METHOD contains : BOOL //check contents, not pointer value
VAR_INPUT
	value : REFERENCE TO AdsMessage;
END_VAR
VAR_OUTPUT
	atIndex : INT;
END_VAR
VAR
	temp : REFERENCE TO AdsMessage;
	i : INT;
END_VAR
IF length = 0 THEN
	contains := FALSE;
	RETURN;
END_IF

FOR i:=0 TO length-1 BY 1 DO
	temp := get(index := i, getSize => );
	
	IF 
		SIZEOF(value) = entrySize AND //same size
		MEMCMP(ADR(temp), ADR(value), SIZEOF(entrySize)) = 0 //same data
	THEN
		contains := TRUE;
		atIndex := i;
		RETURN;
	END_IF
	
END_FOR
contains := FALSE;
END_METHOD

METHOD get : REFERENCE TO AdsMessage
VAR_INPUT
	index : INT;
END_VAR
VAR_OUTPUT
	getSize : UDINT;
	ok : BOOL;
END_VAR
VAR
	temp : POINTER TO AdsMessage;
END_VAR
IF
	length = 0 OR
	index < 0 OR
	index >= length
THEN
	RETURN;
END_IF

ok := elements.GetEntry(diIndex := index, pResultEntry := ADR(temp));
get REF= temp^;

getSize := SIZEOF(get);
END_METHOD

METHOD isEmpty : BOOL
VAR_INPUT
END_VAR
isEmpty := length = 0;
END_METHOD

METHOD poll : AdsMessage
VAR_OUTPUT
	getSize : ULINT;
END_VAR
VAR
	tempRef : REFERENCE TO AdsMessage;
	tempPtr : POINTER TO AdsMessage;
END_VAR
IF length > 0 THEN
	tempRef REF= get(index := 0, getSize => getSize);
	//poll := get(index := 0, getSize => getSize);
	poll := tempRef;
	
	tempPtr := ADR(tempRef);
	__DELETE(tempPtr);
	
	elements.RemoveEntry(diIndex := 0);
	
	length := length - 1;
END_IF
END_METHOD

METHOD push : BOOL
VAR_INPUT
	value : REFERENCE TO AdsMessage;
END_VAR
VAR
	temp : POINTER TO AdsMessage;
END_VAR
IF length < maxElements THEN
	temp := __NEW(AdsMessage);
	temp^ := value;
	
	push := elements.AddEntryPtr(pEntry := temp);
	
	length := length + 1;
END_IF
END_METHOD

METHOD set : BOOL
VAR_INPUT
	i : INT;
	value : REFERENCE TO AdsMessage;
END_VAR
VAR
	temp : REFERENCE TO AdsMessage;
END_VAR
IF length = 0 THEN
	RETURN;
END_IF

IF i >= 0 AND i < length THEN
	temp REF= get(i);
	temp := value;
	
	set := TRUE;
END_IF
END_METHOD

{attribute 'call_after_init'}
METHOD setup : BOOL
VAR_INPUT
END_VAR
entrySize := SIZEOF(AdsMessage);

clear();
END_METHOD

METHOD size : INT
size := length;
END_METHOD

END_FUNCTION_BLOCK

// ---- DUTs/Hardware/Conveyors/ConveyorSC_NC.TcPOU
FUNCTION_BLOCK ConveyorSC_NC
VAR_INPUT
	bEnable : BOOL;
END_VAR
VAR_OUTPUT
	sensorEntry AT %I* : BOOL := TRUE;
	sensorExit AT %I* : BOOL;
	
	trueMode : ConveyorMode;
	requestedMode : ConveyorMode;
	
	position : LREAL;
	velocity : LREAL;
	ready : BOOL;
	error : BOOL;
END_VAR
VAR
	axis : AXIS_REF;
	
	mcReadPosition : MC_ReadActualPosition; //continuous enable FBs
	mcReadVelocity : MC_ReadActualVelocity;
	mcReadError : MC_ReadAxisError;
	mcPower : MC_Power;
	
	mcReset : MC_Reset; //rising edge FBs
	mcMoveAbsolute : MC_MoveAbsolute;
	mcMoveRelative : MC_MoveRelative;
	mcMoveVelocity : MC_MoveVelocity;
	
	mcSetPosition : MC_SetPosition;
	mcStop : MC_Stop;
END_VAR
VAR_STAT CONSTANT
	targetingVelocity : INT := 500;
	continuousVelocity : INT := 100;
END_VAR
(*
standard slat conveyor - no lifter
compliant with PLCopen motion control
*)

blocks();

mcReset.Execute := FALSE;
mcMoveAbsolute.Execute := FALSE;
mcMoveRelative.Execute := FALSE;
mcMoveVelocity.Execute := FALSE;
mcSetPosition.Execute := FALSE;
mcStop.Execute := FALSE;

blocks();

PROPERTY Active : BOOL
GET
Active := 
	mcMoveAbsolute.Busy OR 
	mcMoveRelative.Busy OR 
	mcMoveVelocity.Busy OR 
	mcSetPosition.Busy OR 
	mcReset.Busy OR 
	mcStop.Busy;
END_GET
END_PROPERTY

METHOD PRIVATE blocks : BOOL
mcReadPosition(
	Axis:= axis, 
	Enable:= TRUE, 
	Valid=> , 
	Busy=> , 
	Error=> , 
	ErrorID=> , 
	Position=> position);
	
mcReadVelocity(
	Axis:= axis, 
	Enable:= TRUE, 
	Valid=> , 
	Busy=> , 
	Error=> , 
	ErrorID=> , 
	ActualVelocity=> velocity);
	
mcReadError(
	Axis:= axis, 
	Enable:= TRUE, 
	Valid=> , 
	Busy=> , 
	Error=> , 
	ErrorID=> , 
	AxisErrorID=> );

mcReset(
	Axis:= axis, 
	Execute:= , 
	Done=> , 
	Busy=> , 
	Error=> , 
	ErrorID=> );

mcPower(
	Axis:= axis, 
	Enable:= bEnable, 
	Enable_Positive:= TRUE, 
	Enable_Negative:= TRUE, 
	Override:= 100, 
	BufferMode:= , 
	Options:= , 
	Status=> , 
	Busy=> , 
	Active=> , 
	Error=> , 
	ErrorID=> );

mcMoveAbsolute(
	Axis:= axis, 
	Execute:= , 
	Position:= , 
	Velocity:= targetingVelocity, 
	Acceleration:= , 
	Deceleration:= , 
	Jerk:= , 
	BufferMode:= , 
	Options:= , 
	Done=> , 
	Busy=> , 
	Active=> , 
	CommandAborted=> , 
	Error=> , 
	ErrorID=> );
	
mcMoveRelative(
	Axis:= axis, 
	Execute:= , 
	Distance:= ,
	Velocity:= targetingVelocity, 
	Acceleration:= , 
	Deceleration:= , 
	Jerk:= , 
	BufferMode:= , 
	Options:= , 
	Done=> , 
	Busy=> , 
	Active=> , 
	CommandAborted=> , 
	Error=> , 
	ErrorID=> );
	
mcMoveVelocity( //stopped with stop();
	Axis:= axis, 
	Execute:= , 
	Velocity:= continuousVelocity, 
	Acceleration:= , 
	Deceleration:= , 
	Jerk:= , 
	Direction:= , 
	BufferMode:= , 
	Options:= , 
	InVelocity=> , 
	Busy=> , 
	Active=> , 
	CommandAborted=> , 
	Error=> , 
	ErrorID=> );
	
mcSetPosition(
	Axis:= axis, 
	Execute:= , 
	Position:= , 
	Mode:= , 
	Options:= , 
	Done=> , 
	Busy=> , 
	Error=> , 
	ErrorID=> );
	
mcStop(
	Axis:= axis, 
	Execute:= , 
	Deceleration:= , 
	Jerk:= , 
	Options:= , 
	Done=> , 
	Busy=> , 
	Active=> , 
	CommandAborted=> , 
	Error=> , 
	ErrorID=> );
END_METHOD

PROPERTY CurrentPosition : LREAL
GET
CurrentPosition := position;
END_GET
SET
position := CurrentPosition;
END_SET
END_PROPERTY

{attribute 'monitoring' := 'call'}
PROPERTY IsOccupied : BOOL
GET
IsOccupied := sensorExit OR sensorEntry;
END_GET
END_PROPERTY

METHOD moveAbsolute : BOOL
VAR_INPUT
	newTarget : REAL;
END_VAR
IF NOT Active AND NOT error THEN
	mcMoveAbsolute.Position := newTarget;
	mcMoveAbsolute.Execute := TRUE;
END_IF

moveAbsolute := (*mcMoveAbsolute.Done AND mcMoveAbsolute.Active;*)
	position = newTarget;
END_METHOD

METHOD reset : BOOL
VAR_INPUT
END_VAR
mcReset.Execute := TRUE;

reset := mcReset.Done;
END_METHOD

METHOD setMode : BOOL
VAR_INPUT
	mode : ConveyorMode;
END_VAR
trueMode := mode;
END_METHOD

METHOD setRequest : BOOL
VAR_INPUT
	newRequest : ConveyorMode;
END_VAR
requestedMode := newRequest;
END_METHOD

PROPERTY TargetPosition : LREAL
GET
END_GET
SET
moveAbsolute(newTarget := TargetPosition);
END_SET
END_PROPERTY

END_FUNCTION_BLOCK

// ---- HARDWARE_DISTRUBUTION/A24_A26.TcPOU
FUNCTION_BLOCK A24_A26 EXTENDS GenericSubarea
VAR_IN_OUT
	spacerRecollector : SpacerRecollectionUnit;
END_VAR
VAR
	robot7 : RobotA26;
	robotSliderA26 : ServoNC;
END_VAR
VAR //sensors to detect spacer on transfer conveyors
	spacerPresent_A24_LRC_C02 AT %I* : BOOL;
	spacerPresent_A24_LRC_C04 AT %I* : BOOL;
	spacerPresent_A24_LRC_C06 AT %I* : BOOL;
	spacerPresent_A24_LRC_C08 AT %I* : BOOL;
	spacerPresent_A24_LRC_C10 AT %I* : BOOL;
	spacerPresent_A24_LRC_C12 AT %I* : BOOL;
END_VAR
VAR
	conveyors : ARRAY[1..6] OF POINTER TO Conveyor;
	step : (IDLE, RECEIVE, MEASURE, SEND, VACANT); //idle, align, active, discharge, complete - replacable with SectionTask enum
	step2 : SectionTask;
END_VAR
(*
A2.4 and A2.6 have interdependent processes
this is a prototype FB that contains the data for both subareas
*)

SUPER^();

CASE step OF
	IDLE:
		allConveyorsRequest(newRequest := ConveyorMode.IDLE);
		
		IF TRUE (*incoming bundle*) THEN
			step := RECEIVE;
		END_IF
		
	RECEIVE:
		allConveyorsRequest(newRequest := ConveyorMode.STOP);
		
		IF TRUE (*area 3 is done transferring*) THEN
			step := MEASURE;
		END_IF
		
	MEASURE:
		
		
	SEND:
		allConveyorsRequest(newRequest := ConveyorMode.FORWARD);
		
		IF allConveyorsVacant() THEN
			step := VACANT;
		END_IF
		
	VACANT:
		allConveyorsRequest(newRequest := ConveyorMode.IDLE);
		step := 0;
		
END_CASE

METHOD PROTECTED allConveyorsRequest : BOOL
VAR_INPUT
	newRequest : ConveyorMode;
END_VAR
VAR
	i : INT;
END_VAR
FOR i:=1 TO 6 BY 1 DO
	conveyors[i]^.setRequest(newRequest := newRequest);
END_FOR
END_METHOD

METHOD PROTECTED allConveyorsVacant : BOOL
VAR_INPUT
END_VAR
VAR
	i : INT;
END_VAR
FOR i:=1 TO 6 BY 1 DO
	IF conveyors[i]^.IsOccupied THEN
		RETURN;
	END_IF
END_FOR

allConveyorsVacant := TRUE;
END_METHOD

METHOD PROTECTED callHardware : BOOL
VAR_INPUT
END_VAR
END_METHOD

METHOD PROTECTED runModules : BOOL
VAR_INPUT
END_VAR
// NETWORK 1
END_METHOD

METHOD PROTECTED setupHardware : BOOL
VAR
	i : INT;
END_VAR
conveyors[1] := ADR(ConveyorSyncUnit.A24_LRC_C02);
conveyors[2] := ADR(ConveyorSyncUnit.A24_LRC_C04);
conveyors[3] := ADR(ConveyorSyncUnit.A24_LRC_C06);
conveyors[4] := ADR(ConveyorSyncUnit.A24_LRC_C08);
conveyors[5] := ADR(ConveyorSyncUnit.A24_LRC_C10);
conveyors[6] := ADR(ConveyorSyncUnit.A24_LRC_C12);
END_METHOD

END_FUNCTION_BLOCK

// ---- POUs/Helper Functions/Document/CreateJsonDocumentAuto.TcPOU
PROGRAM CreateJsonDocumentAuto
VAR_INPUT
	visionFrameData : REFERENCE TO VisionFrame;
END_VAR
VAR_OUTPUT
	jsonDocument : STRING(1000); 
END_VAR
VAR
	fbJson : FB_JsonSaxWriter;
	fbJsonDataType : FB_JsonReadWriteDataType;
END_VAR

fbJson.ResetDocument();

fbJsonDataType.AddJsonValueFromSymbol(fbJson, 'VisionFrame', SIZEOF(visionFrameData), ADR(visionFrameData));

fbJson.CopyDocument(jsonDocument, SIZEOF(jsonDocument));

END_PROGRAM

// ---- POUs/Helper Functions/Document/FrameIsValid.TcPOU
FUNCTION FrameIsValid : BOOL
VAR_INPUT
	frame : REFERENCE TO VisionFrame;
END_VAR
VAR
	emptyFrame : VisionFrame;
END_VAR

FrameIsValid := 
	MEMCMP(ADR(frame), ADR(emptyFrame), SIZEOF(VisionFrame)) <> 0 OR
	frame.MaterialID = '' OR
	frame.CheckFor = '' OR
	frame.CameraNumber = 0;

END_FUNCTION

// ---- POUs/Helper Functions/General/WithinTolerance.TcPOU
FUNCTION WithinTolerance : BOOL
VAR_INPUT
	value : LREAL;
	target : LREAL;
	tolerance : LREAL;
END_VAR
(*
checks if value is close enough to target within a given margin
*)

WithinTolerance := ABS(value-target) < tolerance;

END_FUNCTION

// ---- POUs/Helper Functions/Hardware Modules/InsertionQuality.TcPOU
FUNCTION InsertionQuality : BOOL
VAR_IN_OUT
	suctions : ARRAY[*] OF SuctionPad;
END_VAR
VAR_INPUT
	insertionMaterial : STRING;
	recipeMaterial : STRING;
END_VAR
VAR
	i : DINT;
	
	failedPads : INT;
	numPads : INT;
END_VAR

(*
IF insertionMaterial <> recipeMaterial THEN //reintroduce this condition later
	RETURN;
END_IF
*)

FOR i:=LOWER_BOUND(suctions, 1) TO UPPER_BOUND(suctions, 1) BY 1 DO
	IF suctions[i].enable THEN
		numPads := numPads + 1;
		IF NOT suctions[i].occupied THEN
			failedPads := failedPads + 1;
		END_IF
	END_IF
	
END_FOR

InsertionQuality := TRUE;
	//failedPads <= numPads/2;

END_FUNCTION

// ---- POUs/Helper Functions/Material Functions/GetMaterialLength.TcPOU
FUNCTION GetMaterialLength : LREAL
VAR_INPUT
	material : STRING;
END_VAR
VAR
	i : INT;
END_VAR

FOR i:=0 TO CONSTS.numMaterials BY 1 DO
	IF CONSTS.allMaterials[i].code = material THEN
		getMaterialLength := CONSTS.allMaterials[i].length;
		RETURN;
	END_IF
END_FOR
//otherwise, return 0
GetMaterialLength := 0;

END_FUNCTION

// ---- POUs/Helper Functions/Data Manipulation/AddToStringArray.TcPOU
FUNCTION AddToStringArray : BOOL
VAR_IN_OUT
	arr : ARRAY[*] OF STRING; //must start from 0 index
END_VAR
VAR_INPUT
	newString : STRING;
END_VAR
VAR_OUTPUT
	numElements : DINT;
	nextIndex : DINT;
END_VAR
VAR
	i : DINT;
END_VAR

FOR i:=LOWER_BOUND(arr, 1) TO UPPER_BOUND(arr, 1) BY 1 DO	
	IF arr[i] = '' THEN
		arr[i] := newString;
		nextIndex := i + 1;
		AddToStringArray := TRUE;
		EXIT;
	END_IF
	
END_FOR

numElements := UPPER_BOUND(arr, 1) - LOWER_BOUND(arr, 1) + 1;

CleanStringsArray(arr := arr);

END_FUNCTION

// ---- POUs/Helper Functions/Data Manipulation/ArrayContains.TcPOU
FUNCTION ArrayContains : BOOL;
VAR_INPUT
	arr : POINTER TO BYTE;
	arrSize : UDINT;
	element : POINTER TO BYTE;
	typeSize : UDINT;
END_VAR
VAR_OUTPUT
	index : UDINT;
END_VAR
VAR
	i : UDINT;
END_VAR

FOR i:=0 TO arrSize-1 BY typeSize DO
	
	IF MEMCMP(arr[i], element, typeSize) = 0 THEN
		index := i;
		ArrayContains := TRUE;
		RETURN;
	END_IF
	
END_FOR

END_FUNCTION

// ---- POUs/Helper Functions/Data Manipulation/JoinStrings.TcPOU
FUNCTION JoinStrings : STRING
VAR_INPUT
	str1, str2, separator : STRING;
END_VAR
VAR
END_VAR

JoinStrings := CONCAT(str1, separator);
JoinStrings := CONCAT(JoinStrings, str2);

END_FUNCTION
